FUNCTION_BLOCK ABSTRACT FB_Sensor
VAR_INPUT
END_VAR
VAR_OUTPUT
END_VAR
VAR
	{attribute 'OPC.UA.DA' := '1'}
	sensorState : ST_SensorState;
END_VAR

END_FUNCTION_BLOCK

(* stored: Version 1.1.0.1, ProductVersion 3.1.4024.9
   POU FB_Sensor: Id {cd98d21b-bf68-4425-904d-46eec50867b1}, SpecialFunc None *)
